(* CODESYS project crossroad.project

Project tree, tasks and I/O mapping:
  Device : CODESYS Control Win V3, 3S - Smart Software Solutions GmbH, order no. 305021, version 3.5.8.10
    application Application
      libraries: Standard, * (System)
      task MainTask (cyclic, interval t#20ms, priority 1) calls PLC_PRG
      task VISU_TASK (cyclic, interval 100 ms, priority 31) calls VisuElems.Visu_Prg
      program PLC_PRG [CFC]
      visualisation Visualization
  libraries: VisuSymbols, 3.5.8.0 (System)
  text list GlobalTextList
*)

// Device/Application/PLC_PRG
PROGRAM PLC_PRG
VAR
	t1: TOF;
	wlacz1: BOOL;
	zmienna1: TIME;
	zolta1: BOOL;
	czerwona1: BOOL;
	zielona1: BOOL;
	czas: LINT;
	czerwona3: BOOL;
	zielona3: BOOL;
	zolta3: BOOL;
	czerwona2: BOOL;
	zielona2: BOOL;
	zolta2: BOOL;
	zielona4: BOOL;
	zolta4: BOOL;
	czerwona4: BOOL;
	gray1: BOOL;
	yellow1: BOOL;
	zielona5: BOOL;
	zolta5: BOOL;
	czerwona5: BOOL;
	czerwona6: BOOL;
	zielona6: BOOL;
	czerwona7: BOOL;
	zielona7: BOOL;
END_VAR
VAR // added by the converter: edge detectors and wires of the graphical bodies
    _w1, _w2, _w3, _w4, _w6, _w7, _w8, _w9, _w10, _w11, _w12, _w13, _w14, _w15, _w16, _w17, _w18, _w19, _w20, _w21, _w22, _w23, _w24, _w25, _w26, _w27, _w28, _w29, _w30, _w31, _w32, _w33, _w34, _w35, _w36, _w37, _w38, _w39, _w40, _w41, _w42, _w43, _w44, _w45, _w46, _w47, _w48, _w49, _w50, _w51, _w52, _w53, _w54, _w55, _w56, _w57, _w58, _w59, _w60, _w61, _w62, _w63, _w64, _w65, _w66, _w67 : BOOL;
    _w5 : ANY;
END_VAR

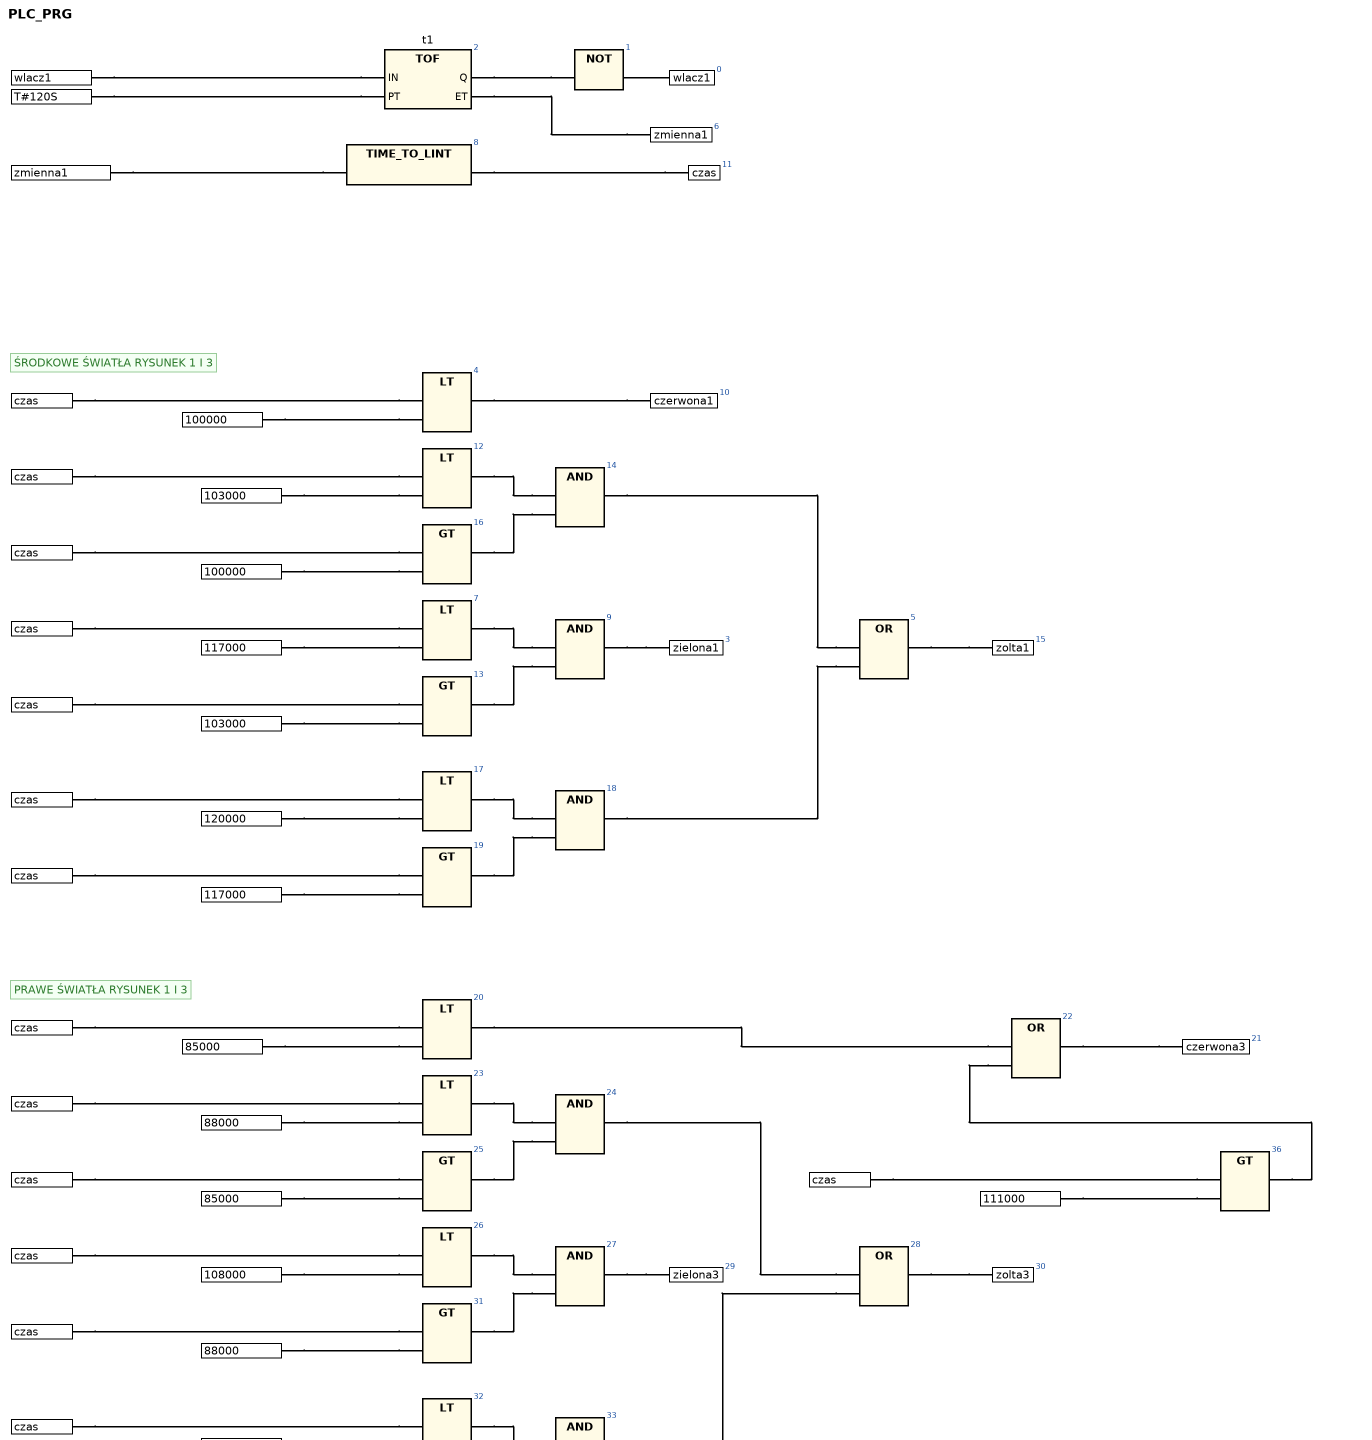
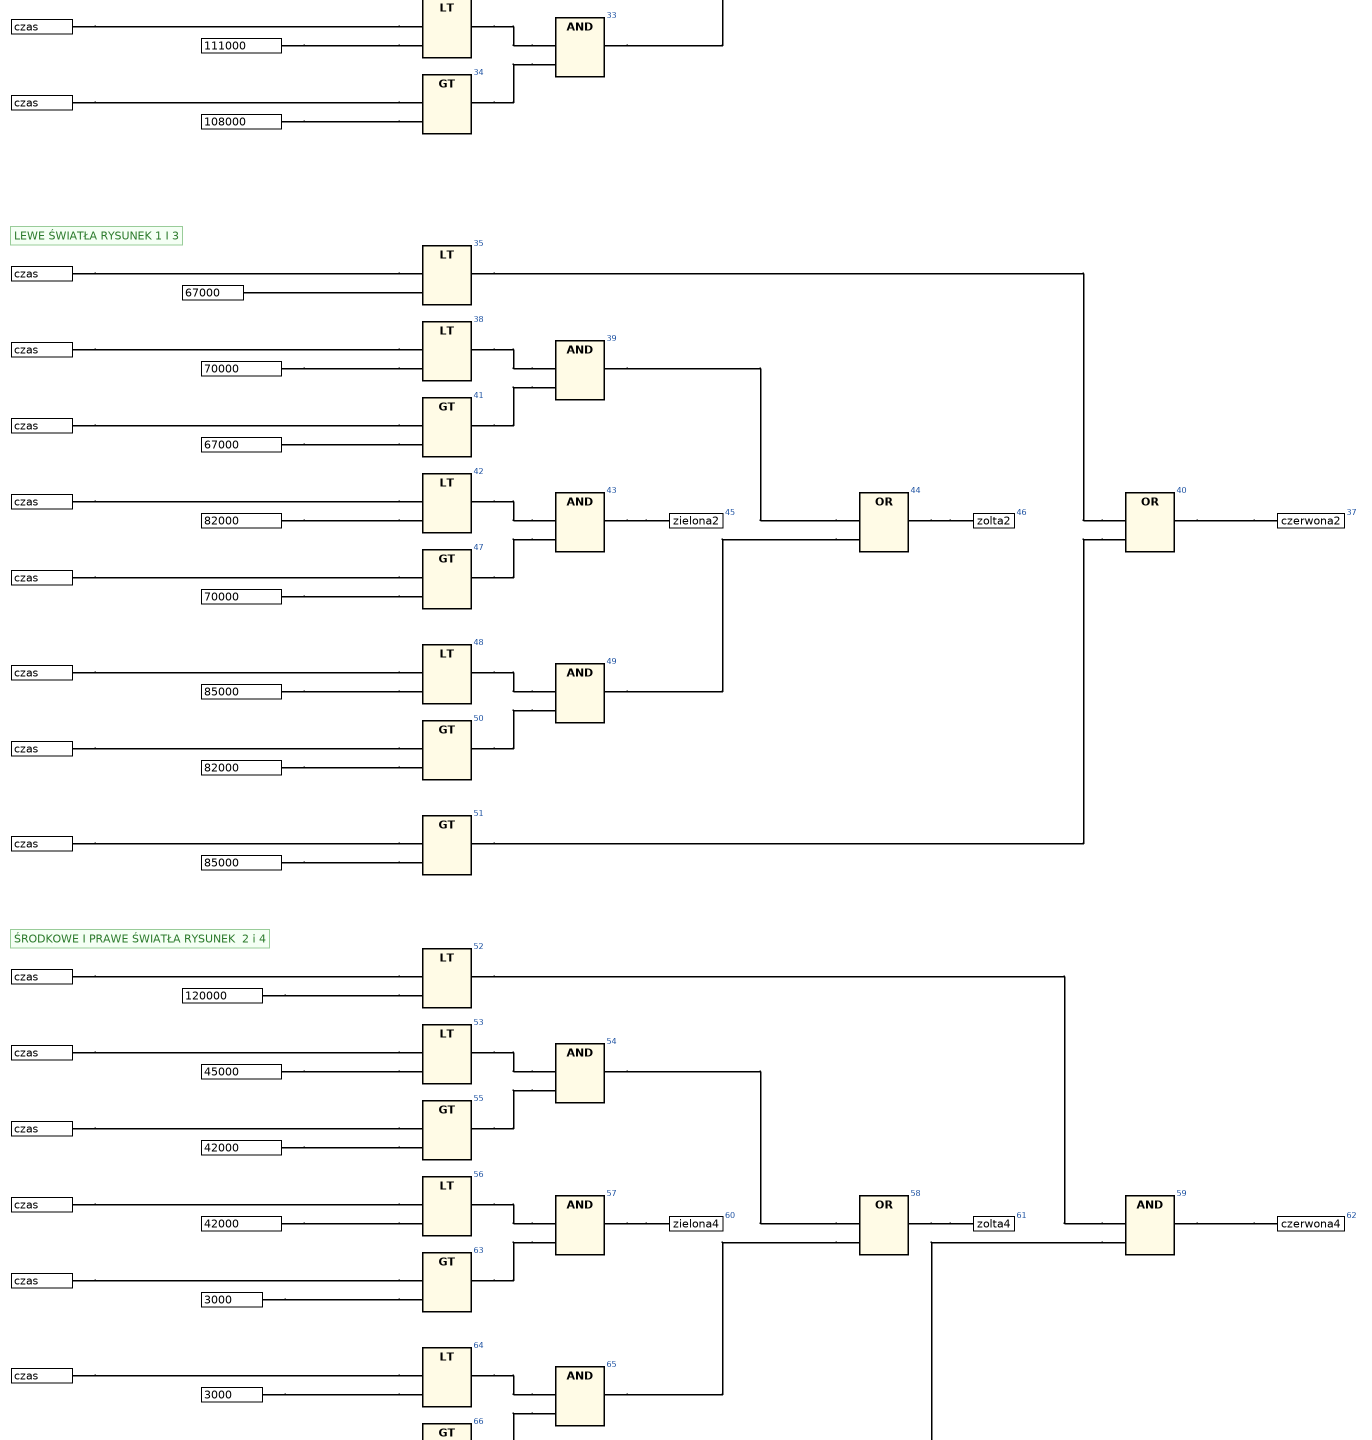
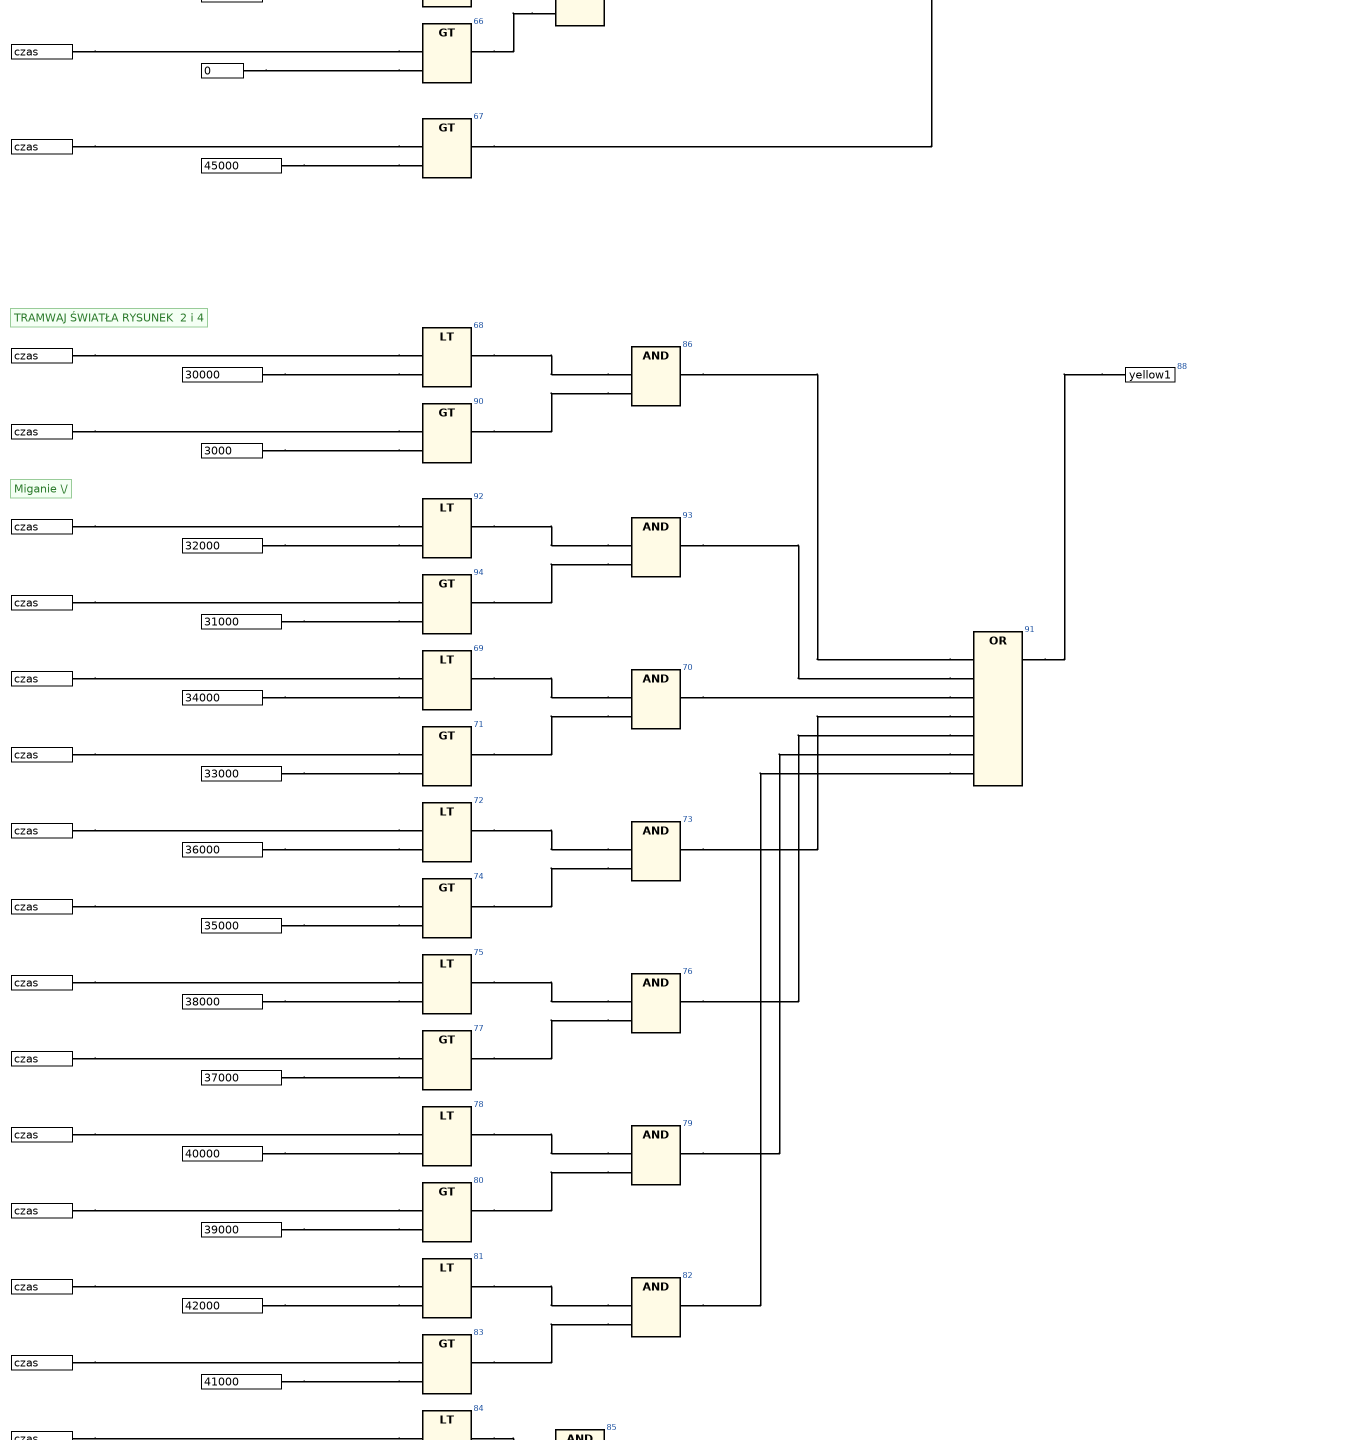
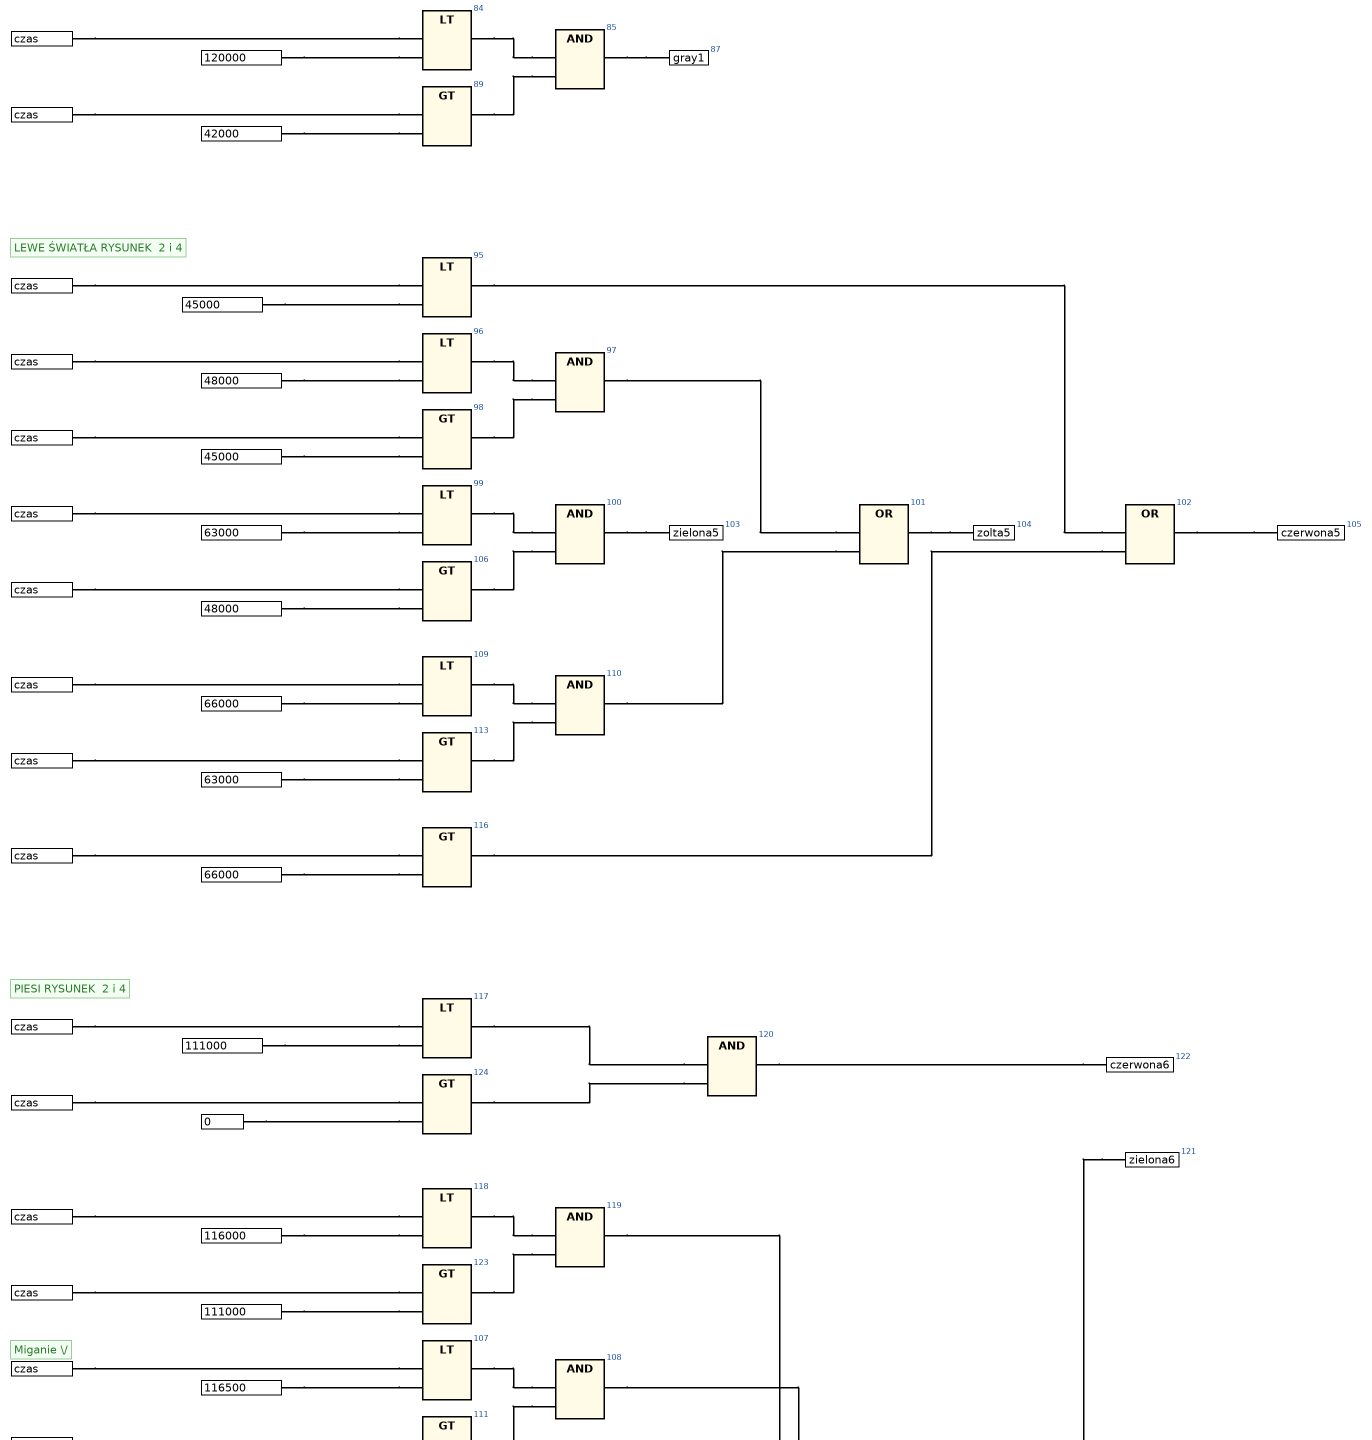
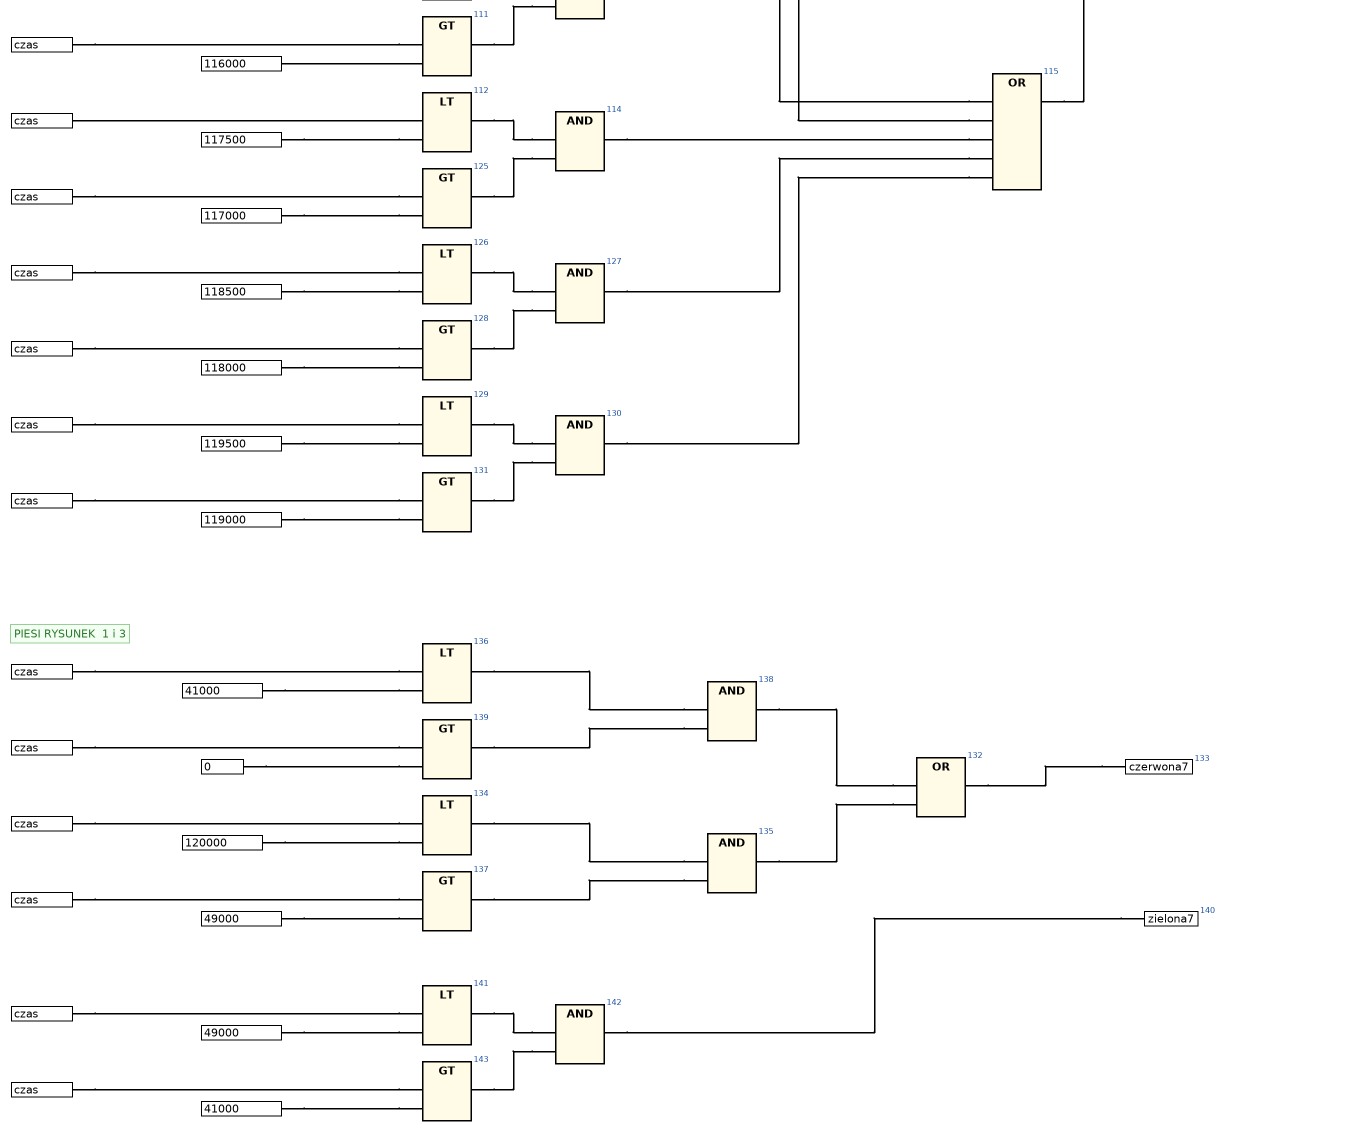
wlacz1 := _w1;
_w1 := NOT t1.Q;
t1(IN := wlacz1, PT := T#120S); // TOF
zielona1 := _w2;
// ŚRODKOWE ŚWIATŁA RYSUNEK 1 I 3
_w5 := _w3 OR _w4;
zmienna1 := t1.ET;
_w2 := czas < 117000 AND _w6;
czerwona1 := czas < 100000;
czas := TIME_TO_LINT(zmienna1);
_w6 := czas > 103000;
_w3 := czas < 103000 AND _w7;
zolta1 := _w5;
_w7 := czas > 100000;
_w4 := czas < 120000 AND _w8;
_w8 := czas > 117000;
// PRAWE ŚWIATŁA RYSUNEK 1 I 3
czerwona3 := _w9;
_w9 := czas < 85000 OR _w10;
_w12 := czas < 88000 AND _w11;
_w11 := czas > 85000;
zielona3 := czas < 108000 AND _w13;
zolta3 := _w12 OR _w14;
_w13 := czas > 88000;
_w14 := czas < 111000 AND _w15;
_w15 := czas > 108000;
// LEWE ŚWIATŁA RYSUNEK 1 I 3
_w10 := czas > 111000;
czerwona2 := _w16;
_w18 := czas < 70000 AND _w17;
_w16 := czas < 67000 OR _w19;
_w17 := czas > 67000;
zielona2 := czas < 82000 AND _w20;
zolta2 := _w18 OR _w21;
_w20 := czas > 70000;
_w21 := czas < 85000 AND _w22;
_w22 := czas > 82000;
_w19 := czas > 85000;
// ŚRODKOWE I PRAWE ŚWIATŁA RYSUNEK  2 i 4
_w24 := czas < 45000 AND _w23;
_w23 := czas > 42000;
zielona4 := czas < 42000 AND _w25;
zolta4 := _w24 OR _w26;
czerwona4 := czas < 120000 AND _w27;
_w25 := czas > 3000;
_w26 := czas < 3000 AND _w28;
_w28 := czas > 0;
_w27 := czas > 45000;
// TRAMWAJ ŚWIATŁA RYSUNEK  2 i 4
_w30 := czas < 34000 AND _w29;
_w29 := czas > 33000;
_w32 := czas < 36000 AND _w31;
_w31 := czas > 35000;
_w34 := czas < 38000 AND _w33;
_w33 := czas > 37000;
_w36 := czas < 40000 AND _w35;
_w35 := czas > 39000;
_w38 := czas < 42000 AND _w37;
_w37 := czas > 41000;
_w41 := czas < 30000 AND _w40;
gray1 := czas < 120000 AND _w39;
yellow1 := _w42;
_w39 := czas > 42000;
_w40 := czas > 3000;
_w42 := _w41 OR _w43 OR _w30 OR _w32 OR _w34 OR _w36 OR _w38;
// Miganie \/
_w43 := czas < 32000 AND _w44;
_w44 := czas > 31000;
// LEWE ŚWIATŁA RYSUNEK  2 i 4
_w46 := czas < 48000 AND _w45;
_w45 := czas > 45000;
zielona5 := czas < 63000 AND _w47;
zolta5 := _w46 OR _w48;
czerwona5 := czas < 45000 OR _w49;
_w47 := czas > 48000;
// Miganie \/
_w51 := czas < 116500 AND _w50;
_w48 := czas < 66000 AND _w52;
_w50 := czas > 116000;
_w52 := czas > 63000;
_w57 := _w54 OR _w51 OR czas < 117500 AND _w53 OR _w55 OR _w56;
_w49 := czas > 66000;
// PIESI RYSUNEK  2 i 4
_w54 := czas < 116000 AND _w58;
zielona6 := _w57;
czerwona6 := czas < 111000 AND _w59;
_w58 := czas > 111000;
_w59 := czas > 0;
_w53 := czas > 117000;
_w55 := czas < 118500 AND _w60;
_w60 := czas > 118000;
_w56 := czas < 119500 AND _w61;
_w61 := czas > 119000;
czerwona7 := _w62 OR _w63;
_w63 := czas < 120000 AND _w64;
// PIESI RYSUNEK  1 i 3
_w64 := czas > 49000;
_w62 := czas < 41000 AND _w65;
_w65 := czas > 0;
zielona7 := _w66;
_w66 := czas < 49000 AND _w67;
_w67 := czas > 41000;

END_PROGRAM

// Device/Application/Visualization
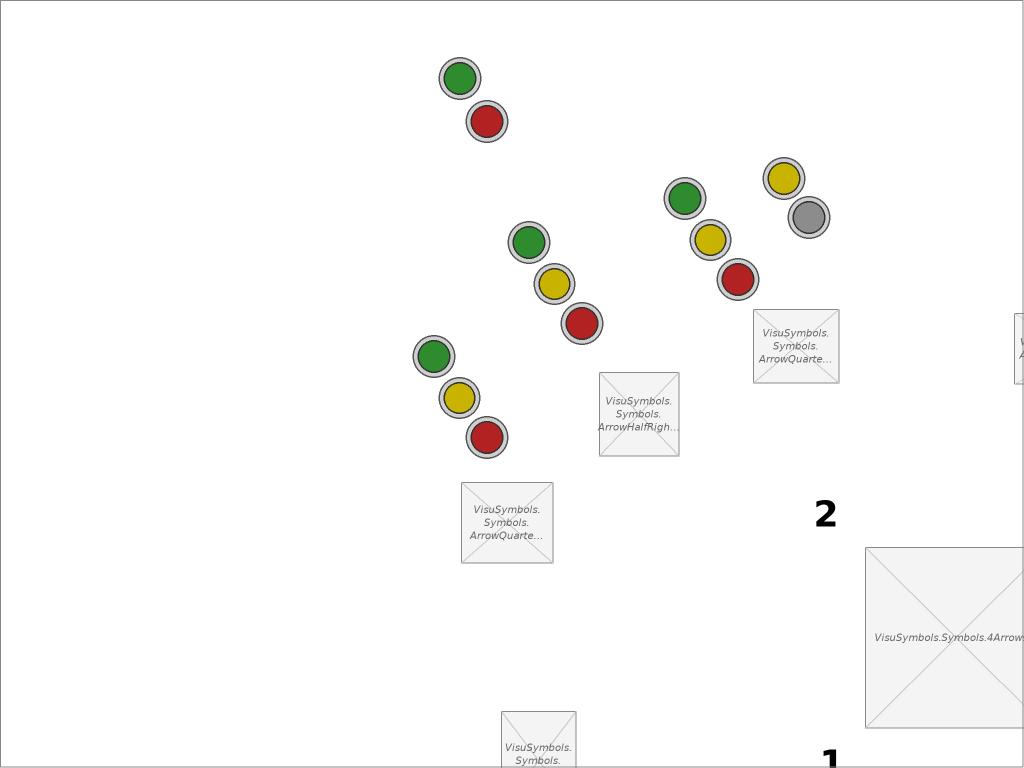
VISUALIZATION Visualization  // 1024x768
    Label (803,742 58x42), "1"
    Label (1024,744 134x50), "4"
    Label (1011,512 159x37), "3"
    Label (751,493 150x42), "2"
    Lamp1 (540,839 56x49), variable: PLC_PRG.czerwona2, style: Lamp-Lamp1-Red
    Lamp1 (540,886 51x48), variable: PLC_PRG.zolta2, style: Lamp-Lamp1-Yellow
    Lamp1 (539,932 50x49), variable: PLC_PRG.zielona2, style: Lamp-Lamp1-Green
    Image (865,547 182x181), image: VisuSymbols.Symbols.4ArrowsIn
    Lamp1 (637,929 56x49), variable: PLC_PRG.czerwona1, style: Lamp-Lamp1-Red
    Lamp1 (637,976 51x48), variable: PLC_PRG.zolta1, style: Lamp-Lamp1-Yellow
    Lamp1 (636,1022 50x49), variable: PLC_PRG.zielona1, style: Lamp-Lamp1-Green
    Lamp1 (737,1015 56x49), variable: PLC_PRG.czerwona3, style: Lamp-Lamp1-Red
    Lamp1 (737,1062 51x48), variable: PLC_PRG.zolta3, style: Lamp-Lamp1-Yellow
    Lamp1 (736,1108 50x49), variable: PLC_PRG.zielona3, style: Lamp-Lamp1-Green
    Lamp1 (1237,291 56x49), variable: PLC_PRG.czerwona1, style: Lamp-Lamp1-Red
    Lamp1 (1265,252 51x48), variable: PLC_PRG.zolta1, style: Lamp-Lamp1-Yellow
    Lamp1 (1292,213 50x49), variable: PLC_PRG.zielona1, style: Lamp-Lamp1-Green
    Lamp1 (1113,1020 56x49), variable: PLC_PRG.czerwona5, style: Lamp-Lamp1-Red
    Lamp1 (1113,1067 51x48), variable: PLC_PRG.zolta5, style: Lamp-Lamp1-Yellow
    Lamp1 (1112,1113 50x49), variable: PLC_PRG.zielona5, style: Lamp-Lamp1-Green
    Lamp1 (1212,959 56x49), variable: PLC_PRG.czerwona4, style: Lamp-Lamp1-Red
    Lamp1 (1212,1006 51x48), variable: PLC_PRG.zolta4, style: Lamp-Lamp1-Yellow
    Lamp1 (1211,1052 50x49), variable: PLC_PRG.zielona4, style: Lamp-Lamp1-Green
    Lamp1 (1294,877 56x49), variable: PLC_PRG.czerwona4, style: Lamp-Lamp1-Red
    Lamp1 (1294,924 51x48), variable: PLC_PRG.zolta4, style: Lamp-Lamp1-Yellow
    Lamp1 (1293,970 50x49), variable: PLC_PRG.zielona4, style: Lamp-Lamp1-Green
    Lamp1 (1113,254 56x49), variable: PLC_PRG.czerwona3, style: Lamp-Lamp1-Red
    Lamp1 (1141,215 51x48), variable: PLC_PRG.zolta3, style: Lamp-Lamp1-Yellow
    Lamp1 (1168,176 50x49), variable: PLC_PRG.zielona3, style: Lamp-Lamp1-Green
    Lamp1 (1316,380 56x49), variable: PLC_PRG.czerwona2, style: Lamp-Lamp1-Red
    Lamp1 (1344,341 51x48), variable: PLC_PRG.zolta2, style: Lamp-Lamp1-Yellow
    Lamp1 (1371,302 50x49), variable: PLC_PRG.zielona2, style: Lamp-Lamp1-Green
    Lamp1 (459,413 56x49), variable: PLC_PRG.czerwona4, style: Lamp-Lamp1-Red
    Lamp1 (434,374 51x48), variable: PLC_PRG.zolta4, style: Lamp-Lamp1-Yellow
    Lamp1 (409,332 50x49), variable: PLC_PRG.zielona4, style: Lamp-Lamp1-Green
    Lamp1 (554,299 56x49), variable: PLC_PRG.czerwona4, style: Lamp-Lamp1-Red
    Lamp1 (529,260 51x48), variable: PLC_PRG.zolta4, style: Lamp-Lamp1-Yellow
    Lamp1 (504,218 50x49), variable: PLC_PRG.zielona4, style: Lamp-Lamp1-Green
    Lamp1 (710,255 56x49), variable: PLC_PRG.czerwona5, style: Lamp-Lamp1-Red
    Lamp1 (685,216 51x48), variable: PLC_PRG.zolta5, style: Lamp-Lamp1-Yellow
    Lamp1 (660,174 50x49), variable: PLC_PRG.zielona5, style: Lamp-Lamp1-Green
    Image (1304,434 101x107), image: VisuSymbols.Symbols.ArrowQuarterLeftRight
    Image (1014,313 125x71), image: VisuSymbols.Symbols.ArrowQuarterRightLeft
    Image (1162,348 87x64), image: VisuSymbols.Symbols.ArrowHalfRightDown
    Image (1310,751 84x102), image: VisuSymbols.Symbols.ArrowQuarterRightRight
    Image (1061,906 75x99), image: VisuSymbols.Symbols.ArrowQuarterLeftLeft
    Image (1136,867 89x71), image: VisuSymbols.Symbols.ArrowHalfLeftUp
    Image (501,711 75x99), image: VisuSymbols.Symbols.ArrowQuarterLeftLeft
    Image (763,895 84x102), image: VisuSymbols.Symbols.ArrowQuarterRightRight
    Image (637,813 84x81), image: VisuSymbols.Symbols.ArrowHalfLeftRight
    Image (599,372 80x84), image: VisuSymbols.Symbols.ArrowHalfRightRight
    Image (461,482 92x81), image: VisuSymbols.Symbols.ArrowQuarterRightDown
    Image (753,309 86x74), image: VisuSymbols.Symbols.ArrowQuarterLeftRight
    Lamp1 (756,154 56x49), variable: PLC_PRG.yellow1, style: Lamp-Lamp1-Yellow
    Lamp1 (781,193 56x49), variable: PLC_PRG.gray1, style: Lamp-Lamp1-Gray
    Lamp1 (1010,1111 56x49), variable: PLC_PRG.yellow1, style: Lamp-Lamp1-Yellow
    Lamp1 (1010,1061 56x49), variable: PLC_PRG.gray1, style: Lamp-Lamp1-Gray
    Lamp1 (383,1066 50x49), variable: PLC_PRG.zielona7, style: Lamp-Lamp1-Green
    Lamp1 (380,1013 56x49), variable: PLC_PRG.czerwona7, style: Lamp-Lamp1-Red
    Lamp1 (435,54 50x49), variable: PLC_PRG.zielona6, style: Lamp-Lamp1-Green
    Lamp1 (459,97 56x49), variable: PLC_PRG.czerwona6, style: Lamp-Lamp1-Red
    Lamp1 (1386,1156 50x49), variable: PLC_PRG.zielona6, style: Lamp-Lamp1-Green
    Lamp1 (1383,1103 56x49), variable: PLC_PRG.czerwona6, style: Lamp-Lamp1-Red
    Lamp1 (1512,129 50x49), variable: PLC_PRG.zielona7, style: Lamp-Lamp1-Green
    Lamp1 (1490,174 56x49), variable: PLC_PRG.czerwona7, style: Lamp-Lamp1-Red
END_VISUALIZATION
